FUNCTION_BLOCK FB_MotionPneumaticActuator_Test EXTENDS TcUnit.FB_TestSuite
VAR
    Expected: BOOL := True;
    Actual: BOOL;
END_VAR

TEST('FB_MotionPneumaticActuator_Test Dummy Test');
AssertEquals(Expected := Expected,
             Actual := Actual,
             Message := 'Error Message');
TEST_FINISHED();

END_FUNCTION_BLOCK

(* stored: Version 1.1.0.1, ProductVersion 3.1.4022.18
   POU FB_MotionPneumaticActuator_Test: Id {69eea798-7b35-4ac7-a85d-de0fbd8448a1}, SpecialFunc None *)
